INTERFACE I_RpcResponseManager

END_INTERFACE

(* stored: Version 1.1.0.1, ProductVersion 3.1.4024.12
   Itf I_RpcResponseManager: Id {d99fa72b-7fb1-42c3-97f3-801a898a58d4} *)
